// ==============================================================================
// FC_HAL_Read - Читання HAL входів через символьні імена
// ==============================================================================
// Project  : Elevator_System
// Author   : Engineering Team
// Version  : 2.0.0
// Generated: 2026-01-14 15:47:36
// ==============================================================================

FUNCTION "FC_HAL_Read" : VOID
{ S7_Optimized_Access := 'TRUE' }
VERSION : 1.0

VAR_IN_OUT
    Redler : ARRAY[*] OF "UDT_Redler";
    Noria  : ARRAY[*] OF "UDT_Noria";
    Gate   : ARRAY[*] OF "UDT_Gate2P";
    Fan    : ARRAY[*] OF "UDT_Fan";
END_VAR

BEGIN
    // ===================================================================
    // REDLERS
    // ===================================================================
    // Редлер_1 (Slot 0, Силос 1, Підвал)
    Redler[0].DI_Speed_OK    := "Redler_1_DI_Speed";
    Redler[0].DI_Breaker_OK  := "Redler_1_DI_Breaker";
    Redler[0].DI_Overflow_OK := "Redler_1_DI_Overflow";

    // Редлер_2 (Slot 1, Силос 2, Підвал)
    Redler[1].DI_Speed_OK    := "Redler_2_DI_Speed";
    Redler[1].DI_Breaker_OK  := "Redler_2_DI_Breaker";
    Redler[1].DI_Overflow_OK := "Redler_2_DI_Overflow";

    // ===================================================================
    // NORIAS
    // ===================================================================
    // Норія_1 (Slot 50, Башта 1)
    Noria[0].DI_Speed_OK      := "Noria_1_DI_Speed";
    Noria[0].DI_Breaker_OK    := "Noria_1_DI_Breaker";
    Noria[0].DI_UpperLevel_OK := "Noria_1_DI_UpperLevel";
    Noria[0].DI_LowerLevel_OK := "Noria_1_DI_LowerLevel";

    // Норія_2 (Slot 51, Башта 2)
    Noria[1].DI_Speed_OK      := "Noria_2_DI_Speed";
    Noria[1].DI_Breaker_OK    := "Noria_2_DI_Breaker";
    Noria[1].DI_UpperLevel_OK := "Noria_2_DI_UpperLevel";
    Noria[1].DI_LowerLevel_OK := "Noria_2_DI_LowerLevel";

    // ===================================================================
    // GATES
    // ===================================================================
    // Засувка_1 (Slot 100, Силос 1, Низ)
    Gate[0].DI_Opened_OK := "Gate_1_DI_Opened";
    Gate[0].DI_Closed_OK := "Gate_1_DI_Closed";

    // Засувка_2 (Slot 101, Силос 2, Низ)
    Gate[1].DI_Opened_OK := "Gate_2_DI_Opened";
    Gate[1].DI_Closed_OK := "Gate_2_DI_Closed";

    // ===================================================================
    // FANS
    // ===================================================================
    // Вентилятор_1 (Slot 150, Силос 1, Верх)
    Fan[0].DI_Breaker_OK := "Fan_1_DI_Breaker";

END_FUNCTION
